// TIA Portal V17 export
FUNCTION "FC_BurnerAlarm" : Void   // FC, LAD
{ S7_Optimized_Access := 'TRUE' }
   VAR_TEMP   // added for the SCL form of the ladder/FBD networks
      _w1 : Bool;
   END_VAR
BEGIN

REGION Network 1: 故障报警：上升沿检测与蜂鸣器置位
   // 7个故障反馈常开触点并联，任意一个接通时经P_TRIG上升沿检测，置位蜂鸣器Q4.7。存储位使用内部数据.报警脉冲。
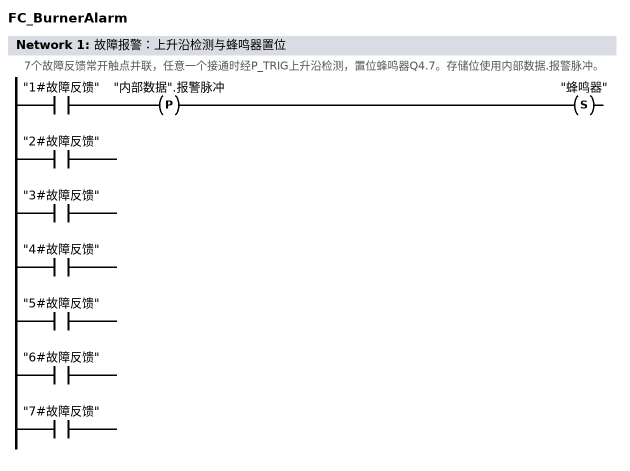
   #_w1 := "1#故障反馈" AND NOT "内部数据".报警脉冲;   // rising edge
   "内部数据".报警脉冲 := "1#故障反馈";
   IF #_w1 THEN "蜂鸣器" := TRUE; END_IF;
END_REGION
END_FUNCTION
